Universal Robots URScript: Bridge_flat_roof_extracted.urscript

def Bridge_flat_roof():
  movej([-1.3958771864520472, -1.5917569599547328, -1.5353903770446777, -1.600466867486471, 1.4777843952178955, 14.233271129915508], a=1.3962634015954636, v=1.0471975511965976)
  movej([-1.9276822249041956, -1.4621073466590424, -1.7524876594543457, -1.5002892401865502, 1.573868989944458, 13.849261649439129], a=1.3962634015954636, v=1.0471975511965976)
  movej([-1.9278915564166468, -1.5445247453502198, -2.0403404235839844, -1.1324440699866791, 1.5930118560791016, 13.790333636591228], a=1.3962634015954636, v=1.0471975511965976)
  movej([-1.9274852911578577, -1.4688049715808411, -1.8157469034194946, -1.4328008455089112, 1.5929371118545532, 13.789905317613872], a=1.3962634015954636, v=1.0471975511965976)
  movej([-2.5445242563830774, -1.5651450914195557, -1.0052506923675537, -2.0938016376891078, 1.5276669263839722, 13.026045091936382], a=1.3962634015954636, v=1.0471975511965976)
  movej([-3.287659231816427, -1.6645165882506312, -1.2465338706970215, -1.7947350941100062, 1.581815481185913, 12.316253487263815], a=1.3962634015954636, v=1.0471975511965976)
  movej([-3.2240458170520228, -1.6823574505248011, -1.8384195566177368, -1.2241854828647156, 1.5686359405517578, 12.511401001607076], a=1.3962634015954636, v=1.0471975511965976)
  movej([-3.224032227193014, -1.6929146252074183, -1.8589739799499512, -1.1932079058936615, 1.5686156749725342, 12.511478249226705], a=1.3962634015954636, v=1.0471975511965976)
  movej([-3.2240458170520228, -1.6823574505248011, -1.8384195566177368, -1.2241854828647156, 1.5686359405517578, 12.511401001607076], a=1.3962634015954636, v=1.0471975511965976)
  movej([-3.2230473200427454, -1.6397167644896449, -1.289588212966919, -1.815672060052389, 1.5677464008331299, 12.511130158101217], a=1.3962634015954636, v=1.0471975511965976)
  movej([-2.2168777624713343, -1.4314818543246766, -1.1272145509719849, -1.9514242611327113, 1.6207340955734253, 12.78394831020573], a=1.3962634015954636, v=1.0471975511965976)
  movej([-1.3958771864520472, -1.5917569599547328, -1.5353903770446777, -1.600466867486471, 1.4777843952178955, 14.233271129915508], a=1.3962634015954636, v=1.0471975511965976)
end
